FUNCTION_BLOCK EL1054
VAR
	_io : EL1054_Data;
	{attribute addProperty Name "WcState"}
	_wcState : WcStateInputToggle;
	{attribute addProperty Name "Info data"}
	_infoData : InfoDataBase;
END_VAR

PROPERTY IO : REFERENCE TO EL1054_Data
GET
IO REF= _io;
END_GET
END_PROPERTY

PROPERTY WcState : REFERENCE TO WcStateInputToggle
GET
WcState REF= _wcState;
END_GET
END_PROPERTY

END_FUNCTION_BLOCK

(* stored: Version 1.1.0.1, ProductVersion 3.1.4024.9
   POU EL1054: Id {b40e8a16-2376-0fda-2ebb-d30723bef1cb}, SpecialFunc None
   Property IO: Id {b5049b93-db96-03ac-128a-6c5a4a79068a}
   Get Get: Id {7c0f2b95-573c-0a0d-3de5-5cd99e294b9d}
   Property WcState: Id {e4461aef-7825-0aa4-0b6e-7c4d5553a158}
   Get Get: Id {5eff3c18-2a6d-0a19-2fbb-995917aac1da} *)
